PROGRAM MAIN
VAR
    {attribute 'TcHmiSymbol' := 'true'}
    bColorState : BOOL := TRUE;
    nCounter : INT := 0;
END_VAR


nCounter := nCounter + 1;

IF nCounter > 1000 THEN
    bColorState := NOT bColorState;
    nCounter := 0;
END_IF;

END_PROGRAM

(* stored: Version 1.1.0.1, ProductVersion 3.1.4024.13
   POU MAIN: Id {5f4c501d-1908-4838-b2d1-d152446867ae}, SpecialFunc None *)
